// Mitsubishi GX Works2 project: Trim_Press 20-08-2023_fr   PLC: Q03UDV

PROGRAM MAIN
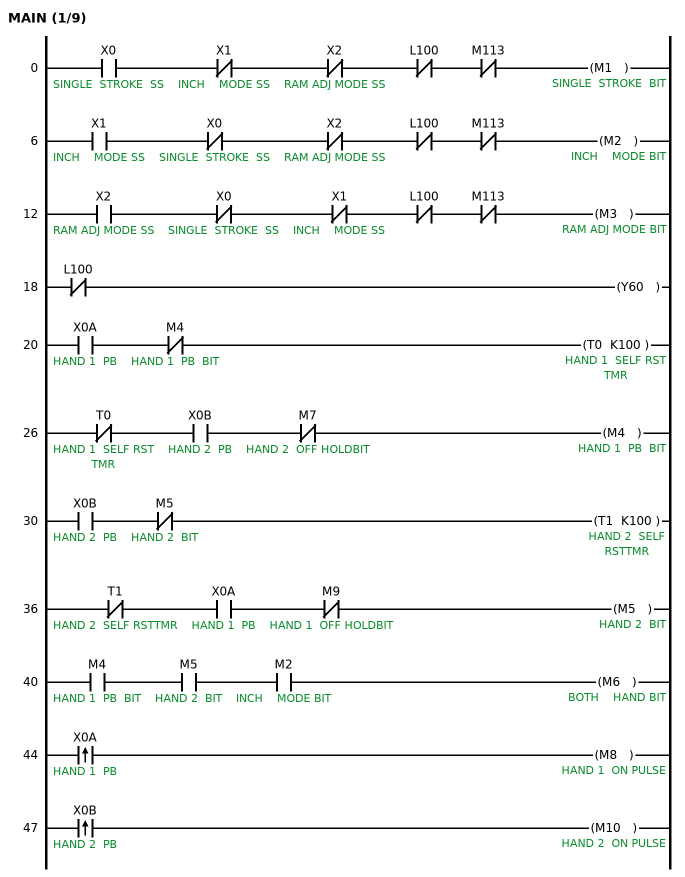
0     LD      X0  ; SINGLE  STROKE  SS
      ANI     X1  ; INCH    MODE SS
      ANI     X2  ; RAM ADJ MODE SS
      ANI     L100
      ANI     M113
      OUT     M1  ; SINGLE  STROKE  BIT
6     LD      X1  ; INCH    MODE SS
      ANI     X0  ; SINGLE  STROKE  SS
      ANI     X2  ; RAM ADJ MODE SS
      ANI     L100
      ANI     M113
      OUT     M2  ; INCH    MODE BIT
12    LD      X2  ; RAM ADJ MODE SS
      ANI     X0  ; SINGLE  STROKE  SS
      ANI     X1  ; INCH    MODE SS
      ANI     L100
      ANI     M113
      OUT     M3  ; RAM ADJ MODE BIT
18    LDI     L100
      OUT     Y60
20    LD      X0A  ; HAND 1  PB
      ANI     M4  ; HAND 1  PB  BIT
      OUT     T0 K100  ; HAND 1  SELF RST TMR
26    LDI     T0  ; HAND 1  SELF RST TMR
      AND     X0B  ; HAND 2  PB
      ANI     M7  ; HAND 2  OFF HOLDBIT
      OUT     M4  ; HAND 1  PB  BIT
30    LD      X0B  ; HAND 2  PB
      ANI     M5  ; HAND 2  BIT
      OUT     T1 K100  ; HAND 2  SELF RSTTMR
36    LDI     T1  ; HAND 2  SELF RSTTMR
      AND     X0A  ; HAND 1  PB
      ANI     M9  ; HAND 1  OFF HOLDBIT
      OUT     M5  ; HAND 2  BIT
40    LD      M4  ; HAND 1  PB  BIT
      AND     M5  ; HAND 2  BIT
      AND     M2  ; INCH    MODE BIT
      OUT     M6  ; BOTH    HAND BIT
44    LDP     X0A  ; HAND 1  PB
      OUT     M8  ; HAND 1  ON PULSE
47    LDP     X0B  ; HAND 2  PB
      OUT     M10  ; HAND 2  ON PULSE
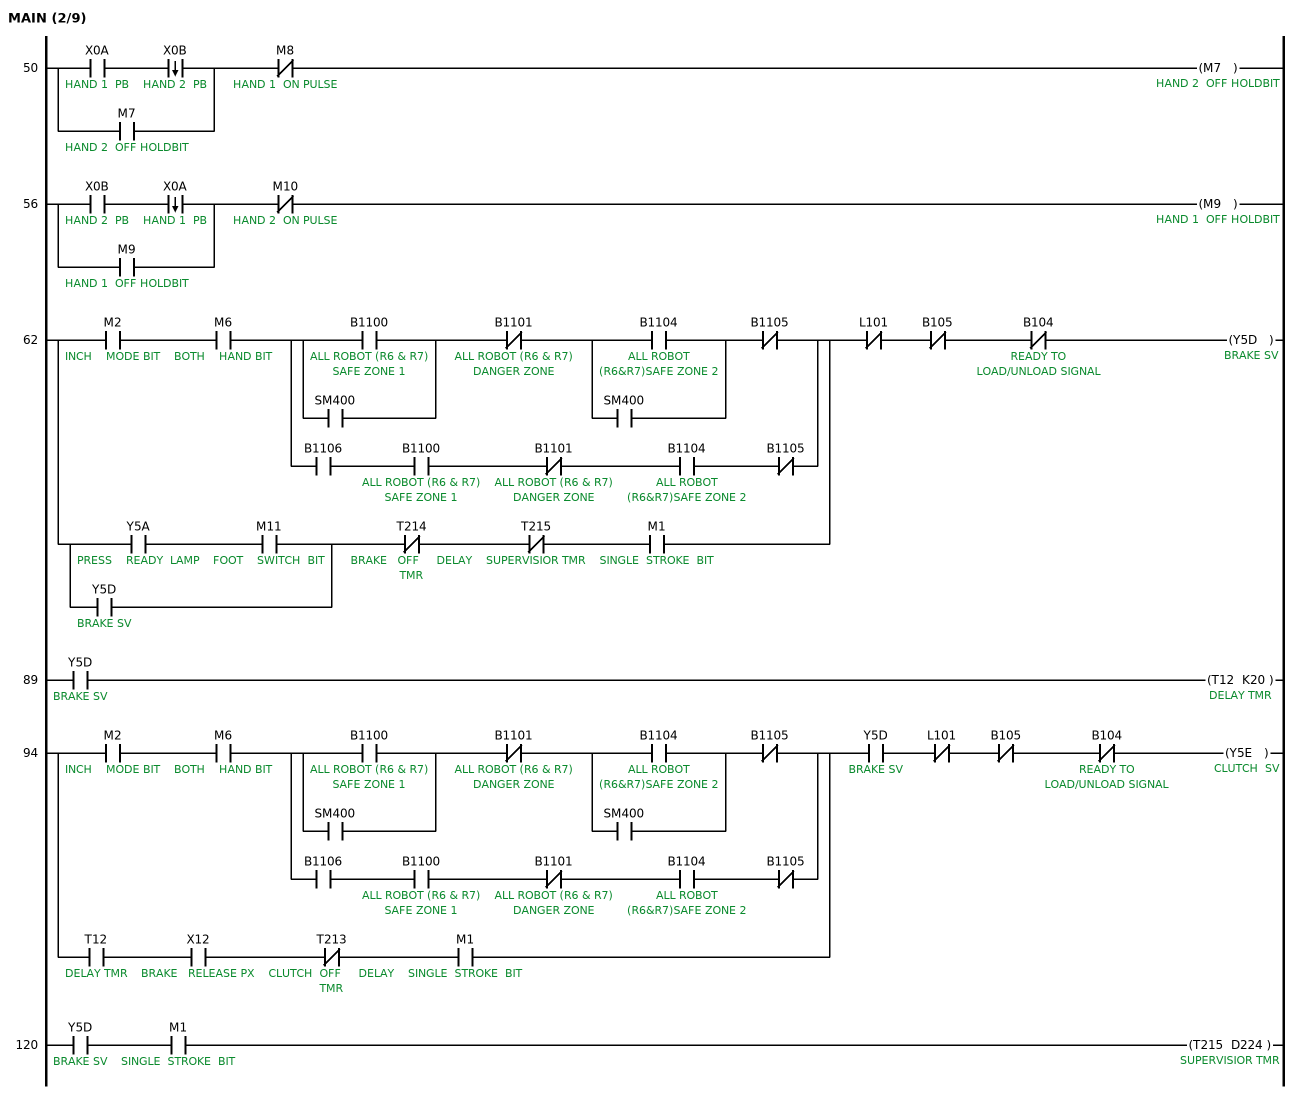
50    LD      X0A  ; HAND 1  PB
      ANDF    X0B  ; HAND 2  PB
      OR      M7  ; HAND 2  OFF HOLDBIT
      ANI     M8  ; HAND 1  ON PULSE
      OUT     M7  ; HAND 2  OFF HOLDBIT
56    LD      X0B  ; HAND 2  PB
      ANDF    X0A  ; HAND 1  PB
      OR      M9  ; HAND 1  OFF HOLDBIT
      ANI     M10  ; HAND 2  ON PULSE
      OUT     M9  ; HAND 1  OFF HOLDBIT
62    LD      M2  ; INCH    MODE BIT
      AND     M6  ; BOTH    HAND BIT
      LD      B1100  ; ALL ROBOT (R6 & R7) SAFE ZONE 1
      OR      SM400
      ANI     B1101  ; ALL ROBOT (R6 & R7) DANGER ZONE
      LD      B1104  ; ALL ROBOT (R6&R7)SAFE ZONE 2
      OR      SM400
      ANB
      ANI     B1105
      LD      B1106
      AND     B1100  ; ALL ROBOT (R6 & R7) SAFE ZONE 1
      ANI     B1101  ; ALL ROBOT (R6 & R7) DANGER ZONE
      AND     B1104  ; ALL ROBOT (R6&R7)SAFE ZONE 2
      ANI     B1105
      ORB
      ANB
      LD      Y5A  ; PRESS    READY  LAMP
      AND     M11  ; FOOT    SWITCH  BIT
      OR      Y5D  ; BRAKE SV
      ANI     T214  ; BRAKE   OFF     DELAY   TMR
      ANI     T215  ; SUPERVISIOR TMR
      AND     M1  ; SINGLE  STROKE  BIT
      ORB
      ANI     L101
      ANI     B105
      ANI     B104  ; READY TO LOAD/UNLOAD SIGNAL
      OUT     Y5D  ; BRAKE SV
89    LD      Y5D  ; BRAKE SV
      OUT     T12 K20  ; DELAY TMR
94    LD      M2  ; INCH    MODE BIT
      AND     M6  ; BOTH    HAND BIT
      LD      B1100  ; ALL ROBOT (R6 & R7) SAFE ZONE 1
      OR      SM400
      ANI     B1101  ; ALL ROBOT (R6 & R7) DANGER ZONE
      LD      B1104  ; ALL ROBOT (R6&R7)SAFE ZONE 2
      OR      SM400
      ANB
      ANI     B1105
      LD      B1106
      AND     B1100  ; ALL ROBOT (R6 & R7) SAFE ZONE 1
      ANI     B1101  ; ALL ROBOT (R6 & R7) DANGER ZONE
      AND     B1104  ; ALL ROBOT (R6&R7)SAFE ZONE 2
      ANI     B1105
      ORB
      ANB
      LD      T12  ; DELAY TMR
      AND     X12  ; BRAKE   RELEASE PX
      ANI     T213  ; CLUTCH  OFF     DELAY   TMR
      AND     M1  ; SINGLE  STROKE  BIT
      ORB
      AND     Y5D  ; BRAKE SV
      ANI     L101
      ANI     B105
      ANI     B104  ; READY TO LOAD/UNLOAD SIGNAL
      OUT     Y5E  ; CLUTCH  SV
120   LD      Y5D  ; BRAKE SV
      AND     M1  ; SINGLE  STROKE  BIT
      OUT     T215 D224  ; SUPERVISIOR TMR
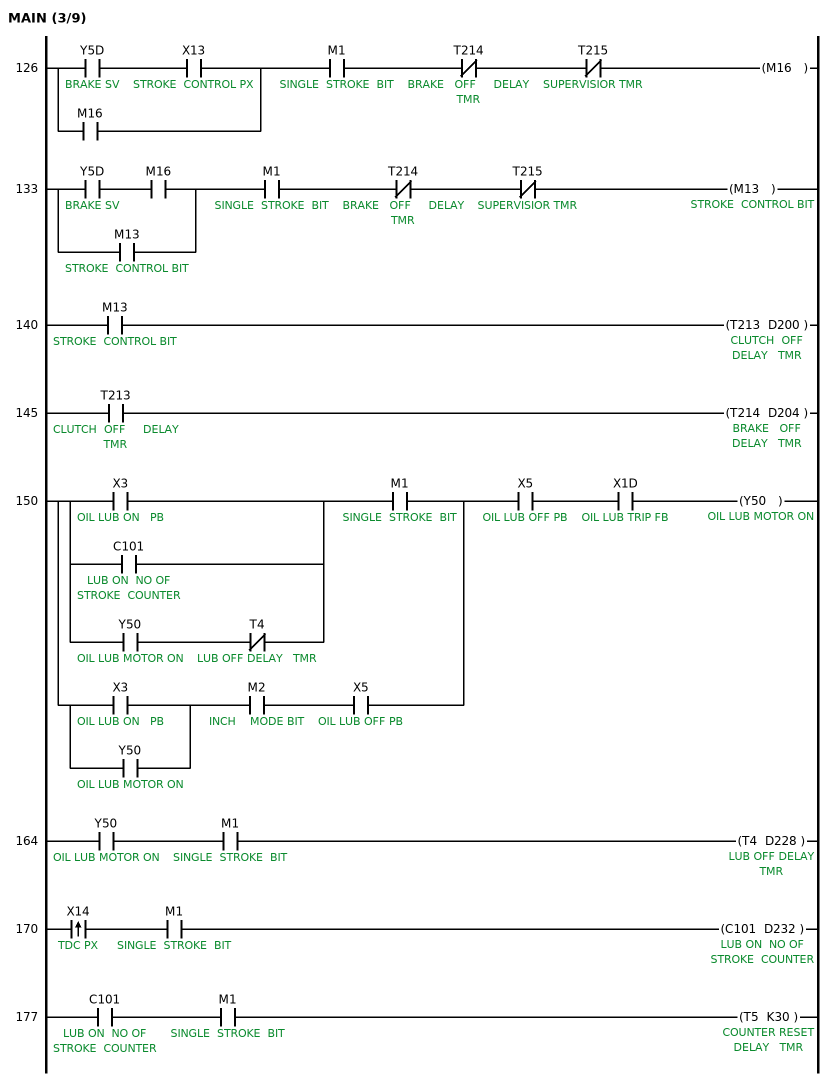
126   LD      Y5D  ; BRAKE SV
      AND     X13  ; STROKE  CONTROL PX
      OR      M16
      AND     M1  ; SINGLE  STROKE  BIT
      ANI     T214  ; BRAKE   OFF     DELAY   TMR
      ANI     T215  ; SUPERVISIOR TMR
      OUT     M16
133   LD      Y5D  ; BRAKE SV
      AND     M16
      OR      M13  ; STROKE  CONTROL BIT
      AND     M1  ; SINGLE  STROKE  BIT
      ANI     T214  ; BRAKE   OFF     DELAY   TMR
      ANI     T215  ; SUPERVISIOR TMR
      OUT     M13  ; STROKE  CONTROL BIT
140   LD      M13  ; STROKE  CONTROL BIT
      OUT     T213 D200  ; CLUTCH  OFF     DELAY   TMR
145   LD      T213  ; CLUTCH  OFF     DELAY   TMR
      OUT     T214 D204  ; BRAKE   OFF     DELAY   TMR
150   LD      X3  ; OIL LUB ON   PB
      OR      C101  ; LUB ON  NO OF   STROKE  COUNTER
      LD      Y50  ; OIL LUB MOTOR ON
      ANI     T4  ; LUB OFF DELAY   TMR
      ORB
      AND     M1  ; SINGLE  STROKE  BIT
      LD      X3  ; OIL LUB ON   PB
      OR      Y50  ; OIL LUB MOTOR ON
      AND     M2  ; INCH    MODE BIT
      AND     X5  ; OIL LUB OFF PB
      ORB
      AND     X5  ; OIL LUB OFF PB
      AND     X1D  ; OIL LUB TRIP FB
      OUT     Y50  ; OIL LUB MOTOR ON
164   LD      Y50  ; OIL LUB MOTOR ON
      AND     M1  ; SINGLE  STROKE  BIT
      OUT     T4 D228  ; LUB OFF DELAY   TMR
170   LDP     X14  ; TDC PX
      AND     M1  ; SINGLE  STROKE  BIT
      OUT     C101 D232  ; LUB ON  NO OF   STROKE  COUNTER
177   LD      C101  ; LUB ON  NO OF   STROKE  COUNTER
      AND     M1  ; SINGLE  STROKE  BIT
      OUT     T5 K30  ; COUNTER RESET   DELAY   TMR
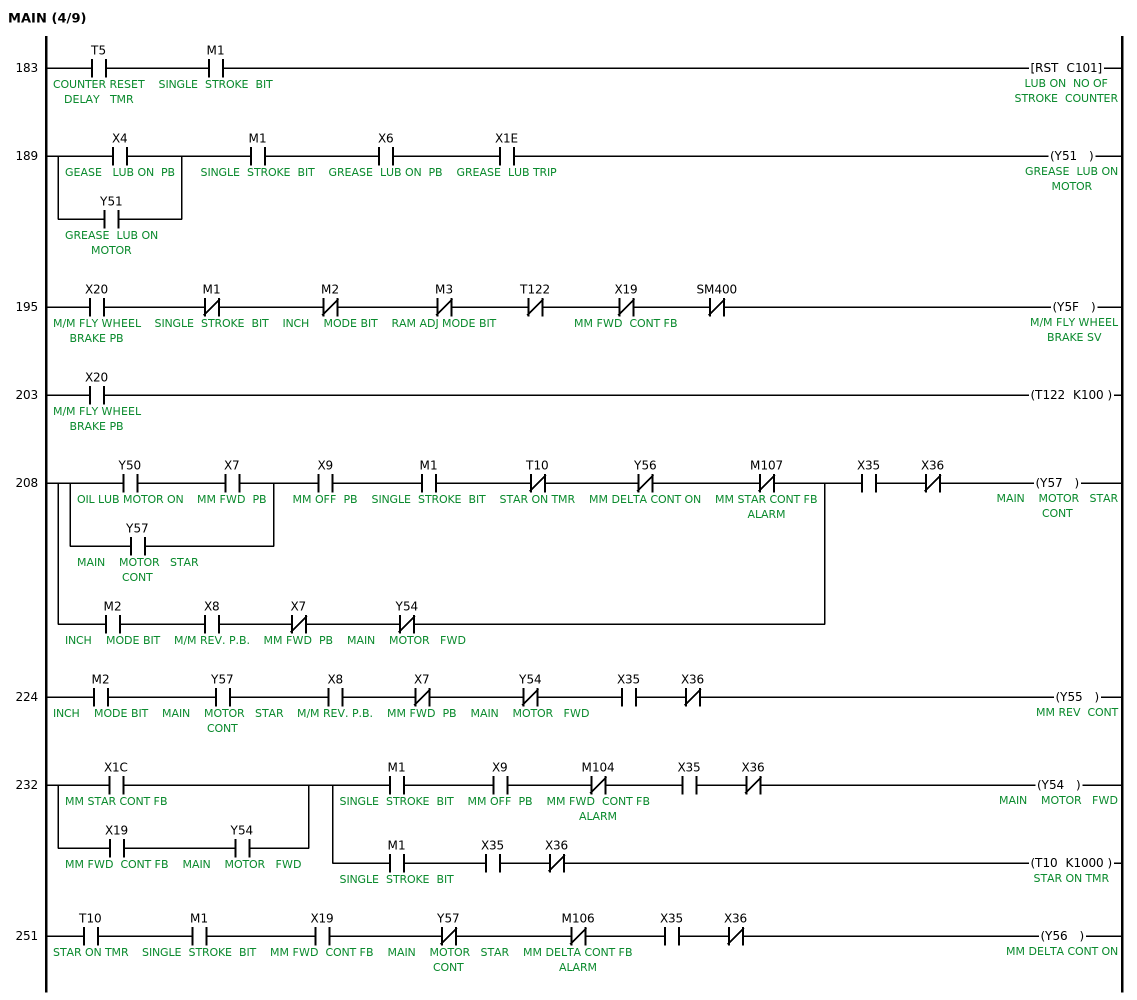
183   LD      T5  ; COUNTER RESET   DELAY   TMR
      AND     M1  ; SINGLE  STROKE  BIT
      RST     C101  ; LUB ON  NO OF   STROKE  COUNTER
189   LD      X4  ; GEASE   LUB ON  PB
      OR      Y51  ; GREASE  LUB ON   MOTOR
      AND     M1  ; SINGLE  STROKE  BIT
      AND     X6  ; GREASE  LUB ON  PB
      AND     X1E  ; GREASE  LUB TRIP
      OUT     Y51  ; GREASE  LUB ON   MOTOR
195   LD      X20  ; M/M FLY WHEEL   BRAKE PB
      ANI     M1  ; SINGLE  STROKE  BIT
      ANI     M2  ; INCH    MODE BIT
      ANI     M3  ; RAM ADJ MODE BIT
      ANI     T122
      ANI     X19  ; MM FWD  CONT FB
      ANI     SM400
      OUT     Y5F  ; M/M FLY WHEEL   BRAKE SV
203   LD      X20  ; M/M FLY WHEEL   BRAKE PB
      OUT     T122 K100
208   LD      Y50  ; OIL LUB MOTOR ON
      AND     X7  ; MM FWD  PB
      OR      Y57  ; MAIN    MOTOR   STAR    CONT
      AND     X9  ; MM OFF  PB
      AND     M1  ; SINGLE  STROKE  BIT
      ANI     T10  ; STAR ON TMR
      ANI     Y56  ; MM DELTA CONT ON
      ANI     M107  ; MM STAR CONT FB ALARM
      LD      M2  ; INCH    MODE BIT
      AND     X8  ; M/M REV. P.B.
      ANI     X7  ; MM FWD  PB
      ANI     Y54  ; MAIN    MOTOR   FWD
      ORB
      AND     X35
      ANI     X36
      OUT     Y57  ; MAIN    MOTOR   STAR    CONT
224   LD      M2  ; INCH    MODE BIT
      AND     Y57  ; MAIN    MOTOR   STAR    CONT
      AND     X8  ; M/M REV. P.B.
      ANI     X7  ; MM FWD  PB
      ANI     Y54  ; MAIN    MOTOR   FWD
      AND     X35
      ANI     X36
      OUT     Y55  ; MM REV  CONT
232   LD      X1C  ; MM STAR CONT FB
      LD      X19  ; MM FWD  CONT FB
      AND     Y54  ; MAIN    MOTOR   FWD
      ORB
      MPS
      AND     M1  ; SINGLE  STROKE  BIT
      AND     X9  ; MM OFF  PB
      ANI     M104  ; MM FWD  CONT FB  ALARM
      AND     X35
      ANI     X36
      OUT     Y54  ; MAIN    MOTOR   FWD
      MPP
      AND     M1  ; SINGLE  STROKE  BIT
      AND     X35
      ANI     X36
      OUT     T10 K1000  ; STAR ON TMR
251   LD      T10  ; STAR ON TMR
      AND     M1  ; SINGLE  STROKE  BIT
      AND     X19  ; MM FWD  CONT FB
      ANI     Y57  ; MAIN    MOTOR   STAR    CONT
      ANI     M106  ; MM DELTA CONT FB ALARM
      AND     X35
      ANI     X36
      OUT     Y56  ; MM DELTA CONT ON
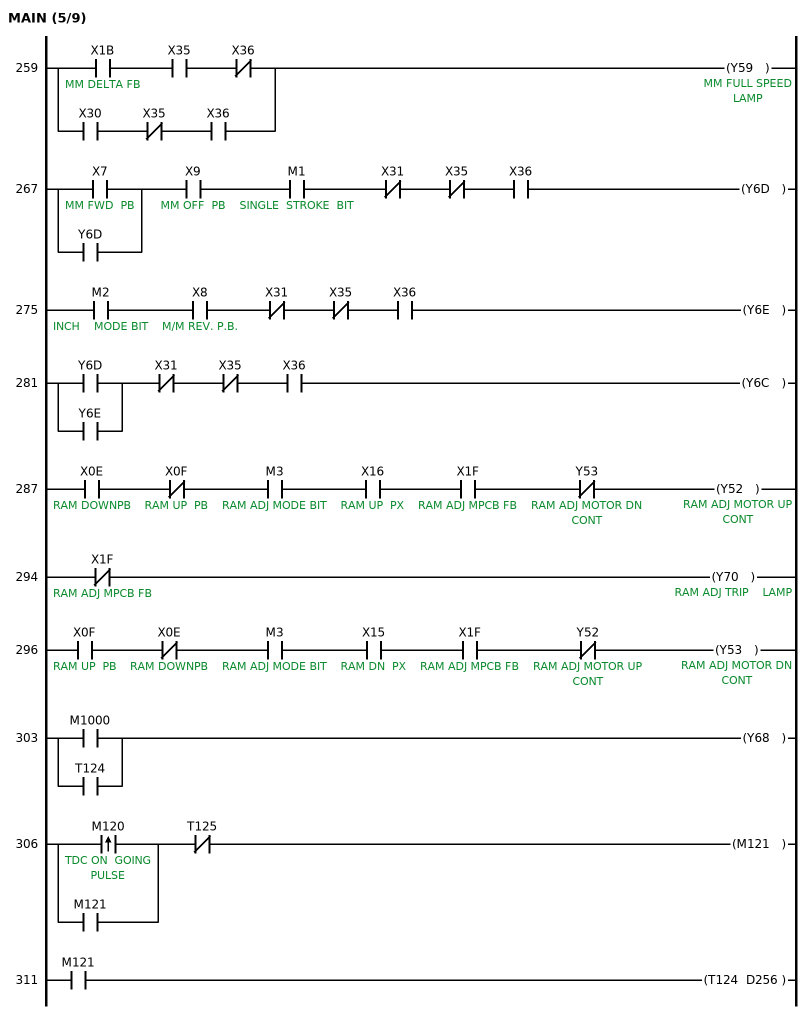
259   LD      X1B  ; MM DELTA FB
      AND     X35
      ANI     X36
      LD      X30
      ANI     X35
      AND     X36
      ORB
      OUT     Y59  ; MM FULL SPEED   LAMP
267   LD      X7  ; MM FWD  PB
      OR      Y6D
      AND     X9  ; MM OFF  PB
      AND     M1  ; SINGLE  STROKE  BIT
      ANI     X31
      ANI     X35
      AND     X36
      OUT     Y6D
275   LD      M2  ; INCH    MODE BIT
      AND     X8  ; M/M REV. P.B.
      ANI     X31
      ANI     X35
      AND     X36
      OUT     Y6E
281   LD      Y6D
      OR      Y6E
      ANI     X31
      ANI     X35
      AND     X36
      OUT     Y6C
287   LD      X0E  ; RAM DOWNPB
      ANI     X0F  ; RAM UP  PB
      AND     M3  ; RAM ADJ MODE BIT
      AND     X16  ; RAM UP  PX
      AND     X1F  ; RAM ADJ MPCB FB
      ANI     Y53  ; RAM ADJ MOTOR DN CONT
      OUT     Y52  ; RAM ADJ MOTOR UP CONT
294   LDI     X1F  ; RAM ADJ MPCB FB
      OUT     Y70  ; RAM ADJ TRIP    LAMP
296   LD      X0F  ; RAM UP  PB
      ANI     X0E  ; RAM DOWNPB
      AND     M3  ; RAM ADJ MODE BIT
      AND     X15  ; RAM DN  PX
      AND     X1F  ; RAM ADJ MPCB FB
      ANI     Y52  ; RAM ADJ MOTOR UP CONT
      OUT     Y53  ; RAM ADJ MOTOR DN CONT
303   LD      M1000
      OR      T124
      OUT     Y68
306   LDP     M120  ; TDC ON  GOING   PULSE
      OR      M121
      ANI     T125
      OUT     M121
311   LD      M121
      OUT     T124 D256
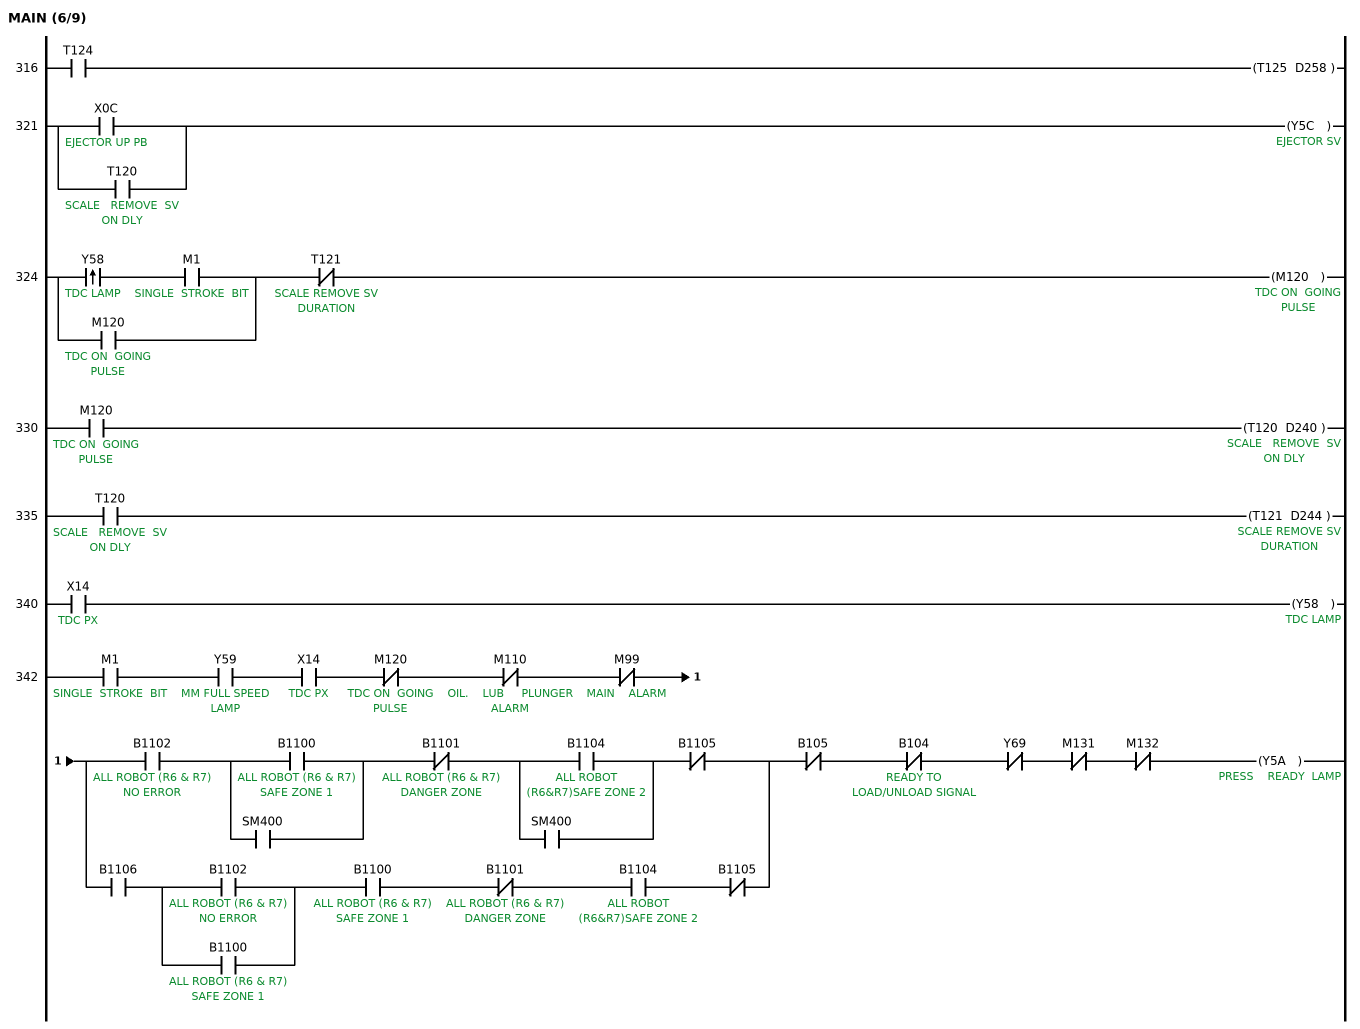
316   LD      T124
      OUT     T125 D258
321   LD      X0C  ; EJECTOR UP PB
      OR      T120  ; SCALE   REMOVE  SV   ON DLY
      OUT     Y5C  ; EJECTOR SV
324   LDP     Y58  ; TDC LAMP
      AND     M1  ; SINGLE  STROKE  BIT
      OR      M120  ; TDC ON  GOING   PULSE
      ANI     T121  ; SCALE REMOVE SV DURATION
      OUT     M120  ; TDC ON  GOING   PULSE
330   LD      M120  ; TDC ON  GOING   PULSE
      OUT     T120 D240  ; SCALE   REMOVE  SV   ON DLY
335   LD      T120  ; SCALE   REMOVE  SV   ON DLY
      OUT     T121 D244  ; SCALE REMOVE SV DURATION
340   LD      X14  ; TDC PX
      OUT     Y58  ; TDC LAMP
342   LD      M1  ; SINGLE  STROKE  BIT
      AND     Y59  ; MM FULL SPEED   LAMP
      AND     X14  ; TDC PX
      ANI     M120  ; TDC ON  GOING   PULSE
      ANI     M110  ; OIL.    LUB     PLUNGER ALARM
      ANI     M99  ; MAIN    ALARM
      LD      B1102  ; ALL ROBOT (R6 & R7) NO ERROR
      LD      B1100  ; ALL ROBOT (R6 & R7) SAFE ZONE 1
      OR      SM400
      ANB
      ANI     B1101  ; ALL ROBOT (R6 & R7) DANGER ZONE
      LD      B1104  ; ALL ROBOT (R6&R7)SAFE ZONE 2
      OR      SM400
      ANB
      ANI     B1105
      LD      B1106
      LD      B1102  ; ALL ROBOT (R6 & R7) NO ERROR
      OR      B1100  ; ALL ROBOT (R6 & R7) SAFE ZONE 1
      ANB
      AND     B1100  ; ALL ROBOT (R6 & R7) SAFE ZONE 1
      ANI     B1101  ; ALL ROBOT (R6 & R7) DANGER ZONE
      AND     B1104  ; ALL ROBOT (R6&R7)SAFE ZONE 2
      ANI     B1105
      ORB
      ANB
      ANI     B105
      ANI     B104  ; READY TO LOAD/UNLOAD SIGNAL
      ANI     Y69
      ANI     M131
      ANI     M132
      OUT     Y5A  ; PRESS    READY  LAMP
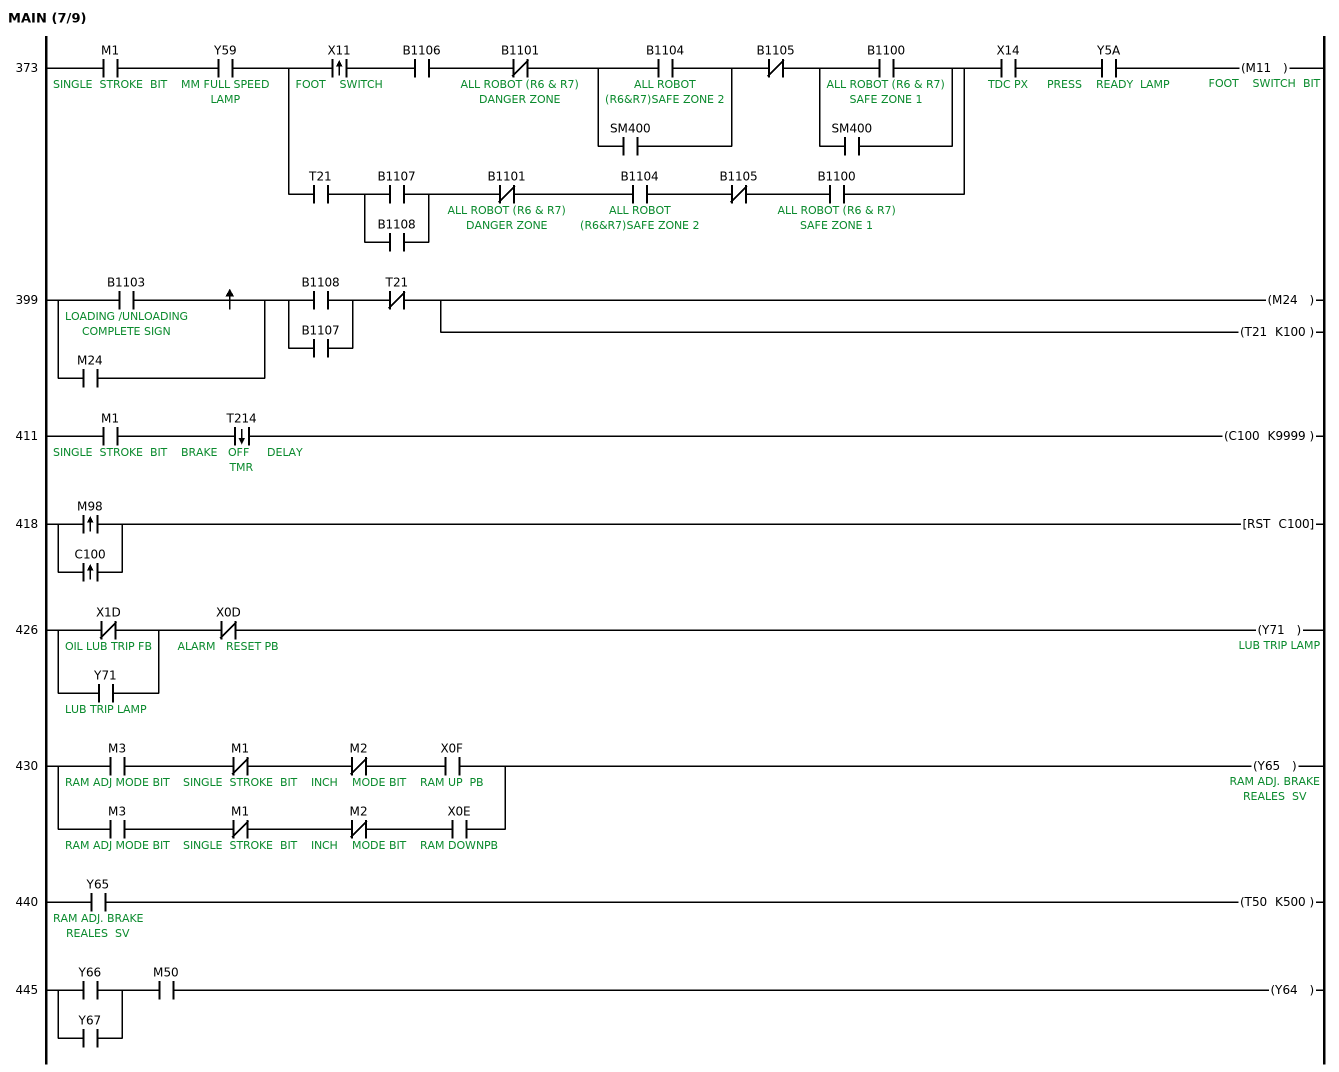
373   LD      M1  ; SINGLE  STROKE  BIT
      AND     Y59  ; MM FULL SPEED   LAMP
      LDP     X11  ; FOOT    SWITCH
      AND     B1106
      ANI     B1101  ; ALL ROBOT (R6 & R7) DANGER ZONE
      LD      B1104  ; ALL ROBOT (R6&R7)SAFE ZONE 2
      OR      SM400
      ANB
      ANI     B1105
      LD      B1100  ; ALL ROBOT (R6 & R7) SAFE ZONE 1
      OR      SM400
      ANB
      LD      T21
      LD      B1107
      OR      B1108
      ANB
      ANI     B1101  ; ALL ROBOT (R6 & R7) DANGER ZONE
      AND     B1104  ; ALL ROBOT (R6&R7)SAFE ZONE 2
      ANI     B1105
      AND     B1100  ; ALL ROBOT (R6 & R7) SAFE ZONE 1
      ORB
      ANB
      AND     X14  ; TDC PX
      AND     Y5A  ; PRESS    READY  LAMP
      OUT     M11  ; FOOT    SWITCH  BIT
399   LD      B1103  ; LOADING /UNLOADING COMPLETE SIGN
      MEP
      OR      M24
      LD      B1108
      OR      B1107
      ANB
      ANI     T21
      OUT     M24
      OUT     T21 K100
411   LD      M1  ; SINGLE  STROKE  BIT
      ANDF    T214  ; BRAKE   OFF     DELAY   TMR
      OUT     C100 K9999
418   LDP     M98
      ORP     C100
      RST     C100
426   LDI     X1D  ; OIL LUB TRIP FB
      OR      Y71  ; LUB TRIP LAMP
      ANI     X0D  ; ALARM   RESET PB
      OUT     Y71  ; LUB TRIP LAMP
430   LD      M3  ; RAM ADJ MODE BIT
      ANI     M1  ; SINGLE  STROKE  BIT
      ANI     M2  ; INCH    MODE BIT
      AND     X0F  ; RAM UP  PB
      LD      M3  ; RAM ADJ MODE BIT
      ANI     M1  ; SINGLE  STROKE  BIT
      ANI     M2  ; INCH    MODE BIT
      AND     X0E  ; RAM DOWNPB
      ORB
      OUT     Y65  ; RAM ADJ. BRAKE  REALES  SV
440   LD      Y65  ; RAM ADJ. BRAKE  REALES  SV
      OUT     T50 K500
445   LD      Y66
      OR      Y67
      AND     M50
      OUT     Y64
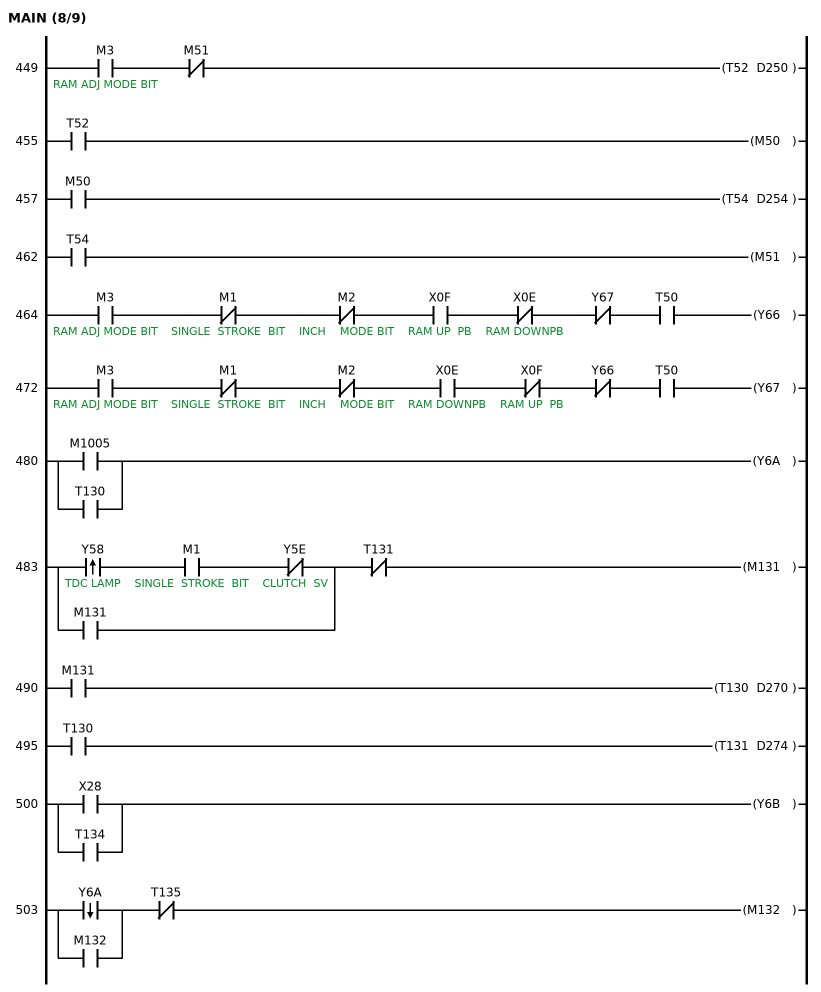
449   LD      M3  ; RAM ADJ MODE BIT
      ANI     M51
      OUT     T52 D250
455   LD      T52
      OUT     M50
457   LD      M50
      OUT     T54 D254
462   LD      T54
      OUT     M51
464   LD      M3  ; RAM ADJ MODE BIT
      ANI     M1  ; SINGLE  STROKE  BIT
      ANI     M2  ; INCH    MODE BIT
      AND     X0F  ; RAM UP  PB
      ANI     X0E  ; RAM DOWNPB
      ANI     Y67
      AND     T50
      OUT     Y66
472   LD      M3  ; RAM ADJ MODE BIT
      ANI     M1  ; SINGLE  STROKE  BIT
      ANI     M2  ; INCH    MODE BIT
      AND     X0E  ; RAM DOWNPB
      ANI     X0F  ; RAM UP  PB
      ANI     Y66
      AND     T50
      OUT     Y67
480   LD      M1005
      OR      T130
      OUT     Y6A
483   LDP     Y58  ; TDC LAMP
      AND     M1  ; SINGLE  STROKE  BIT
      ANI     Y5E  ; CLUTCH  SV
      OR      M131
      ANI     T131
      OUT     M131
490   LD      M131
      OUT     T130 D270
495   LD      T130
      OUT     T131 D274
500   LD      X28
      OR      T134
      OUT     Y6B
503   LDF     Y6A
      OR      M132
      ANI     T135
      OUT     M132
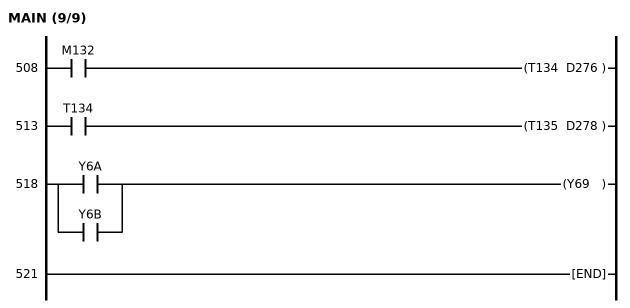
508   LD      M132
      OUT     T134 D276
513   LD      T134
      OUT     T135 D278
518   LD      Y6A
      OR      Y6B
      OUT     Y69
521   END
END_PROGRAM

PROGRAM MAIN01
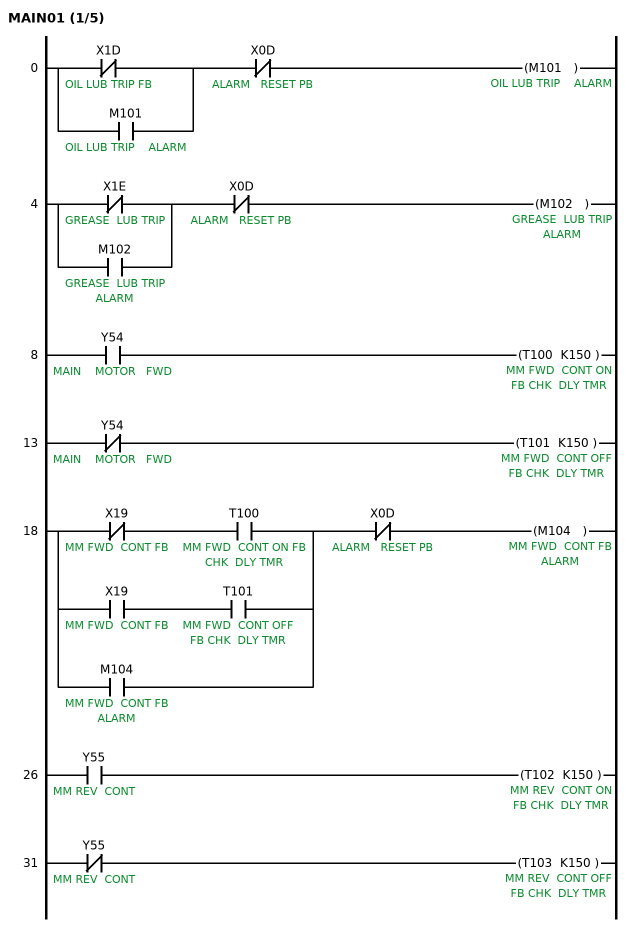
0     LDI     X1D  ; OIL LUB TRIP FB
      OR      M101  ; OIL LUB TRIP    ALARM
      ANI     X0D  ; ALARM   RESET PB
      OUT     M101  ; OIL LUB TRIP    ALARM
4     LDI     X1E  ; GREASE  LUB TRIP
      OR      M102  ; GREASE  LUB TRIP  ALARM
      ANI     X0D  ; ALARM   RESET PB
      OUT     M102  ; GREASE  LUB TRIP  ALARM
8     LD      Y54  ; MAIN    MOTOR   FWD
      OUT     T100 K150  ; MM FWD  CONT ON FB CHK  DLY TMR
13    LDI     Y54  ; MAIN    MOTOR   FWD
      OUT     T101 K150  ; MM FWD  CONT OFF FB CHK  DLY TMR
18    LDI     X19  ; MM FWD  CONT FB
      AND     T100  ; MM FWD  CONT ON FB CHK  DLY TMR
      LD      X19  ; MM FWD  CONT FB
      AND     T101  ; MM FWD  CONT OFF FB CHK  DLY TMR
      ORB
      OR      M104  ; MM FWD  CONT FB  ALARM
      ANI     X0D  ; ALARM   RESET PB
      OUT     M104  ; MM FWD  CONT FB  ALARM
26    LD      Y55  ; MM REV  CONT
      OUT     T102 K150  ; MM REV  CONT ON FB CHK  DLY TMR
31    LDI     Y55  ; MM REV  CONT
      OUT     T103 K150  ; MM REV  CONT OFF FB CHK  DLY TMR
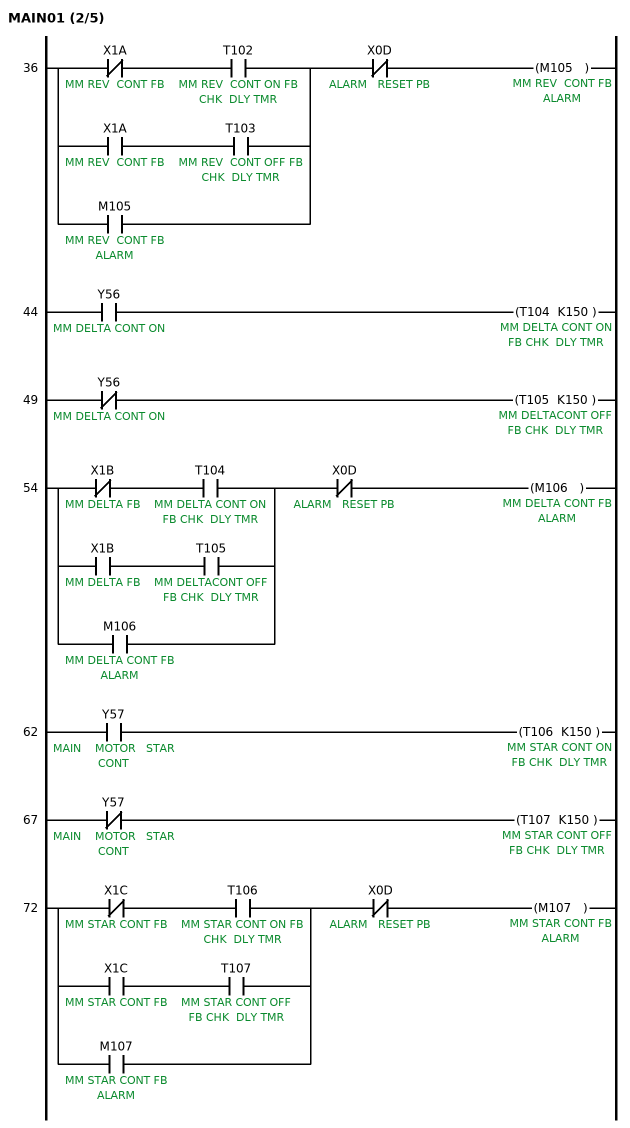
36    LDI     X1A  ; MM REV  CONT FB
      AND     T102  ; MM REV  CONT ON FB CHK  DLY TMR
      LD      X1A  ; MM REV  CONT FB
      AND     T103  ; MM REV  CONT OFF FB CHK  DLY TMR
      ORB
      OR      M105  ; MM REV  CONT FB ALARM
      ANI     X0D  ; ALARM   RESET PB
      OUT     M105  ; MM REV  CONT FB ALARM
44    LD      Y56  ; MM DELTA CONT ON
      OUT     T104 K150  ; MM DELTA CONT ON FB CHK  DLY TMR
49    LDI     Y56  ; MM DELTA CONT ON
      OUT     T105 K150  ; MM DELTACONT OFF FB CHK  DLY TMR
54    LDI     X1B  ; MM DELTA FB
      AND     T104  ; MM DELTA CONT ON FB CHK  DLY TMR
      LD      X1B  ; MM DELTA FB
      AND     T105  ; MM DELTACONT OFF FB CHK  DLY TMR
      ORB
      OR      M106  ; MM DELTA CONT FB ALARM
      ANI     X0D  ; ALARM   RESET PB
      OUT     M106  ; MM DELTA CONT FB ALARM
62    LD      Y57  ; MAIN    MOTOR   STAR    CONT
      OUT     T106 K150  ; MM STAR CONT ON FB CHK  DLY TMR
67    LDI     Y57  ; MAIN    MOTOR   STAR    CONT
      OUT     T107 K150  ; MM STAR CONT OFF FB CHK  DLY TMR
72    LDI     X1C  ; MM STAR CONT FB
      AND     T106  ; MM STAR CONT ON FB CHK  DLY TMR
      LD      X1C  ; MM STAR CONT FB
      AND     T107  ; MM STAR CONT OFF FB CHK  DLY TMR
      ORB
      OR      M107  ; MM STAR CONT FB ALARM
      ANI     X0D  ; ALARM   RESET PB
      OUT     M107  ; MM STAR CONT FB ALARM
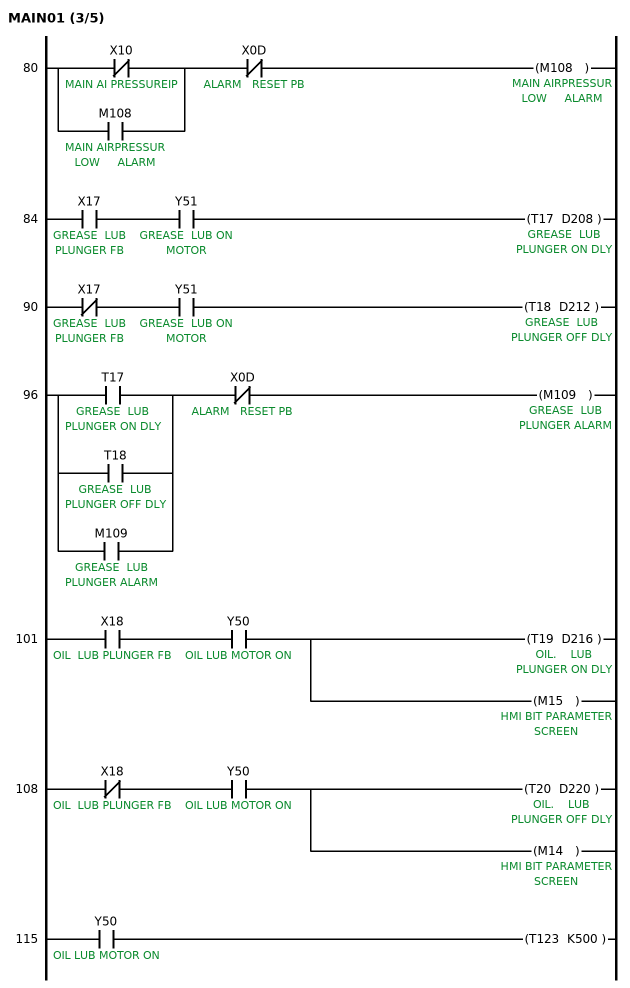
80    LDI     X10  ; MAIN AI PRESSUREIP
      OR      M108  ; MAIN AIRPRESSUR LOW     ALARM
      ANI     X0D  ; ALARM   RESET PB
      OUT     M108  ; MAIN AIRPRESSUR LOW     ALARM
84    LD      X17  ; GREASE  LUB     PLUNGER FB
      AND     Y51  ; GREASE  LUB ON   MOTOR
      OUT     T17 D208  ; GREASE  LUB     PLUNGER ON DLY
90    LDI     X17  ; GREASE  LUB     PLUNGER FB
      AND     Y51  ; GREASE  LUB ON   MOTOR
      OUT     T18 D212  ; GREASE  LUB     PLUNGER OFF DLY
96    LD      T17  ; GREASE  LUB     PLUNGER ON DLY
      OR      T18  ; GREASE  LUB     PLUNGER OFF DLY
      OR      M109  ; GREASE  LUB     PLUNGER ALARM
      ANI     X0D  ; ALARM   RESET PB
      OUT     M109  ; GREASE  LUB     PLUNGER ALARM
101   LD      X18  ; OIL  LUB PLUNGER FB
      AND     Y50  ; OIL LUB MOTOR ON
      OUT     T19 D216  ; OIL.    LUB     PLUNGER ON DLY
      OUT     M15  ; HMI BIT PARAMETER SCREEN
108   LDI     X18  ; OIL  LUB PLUNGER FB
      AND     Y50  ; OIL LUB MOTOR ON
      OUT     T20 D220  ; OIL.    LUB     PLUNGER OFF DLY
      OUT     M14  ; HMI BIT PARAMETER SCREEN
115   LD      Y50  ; OIL LUB MOTOR ON
      OUT     T123 K500
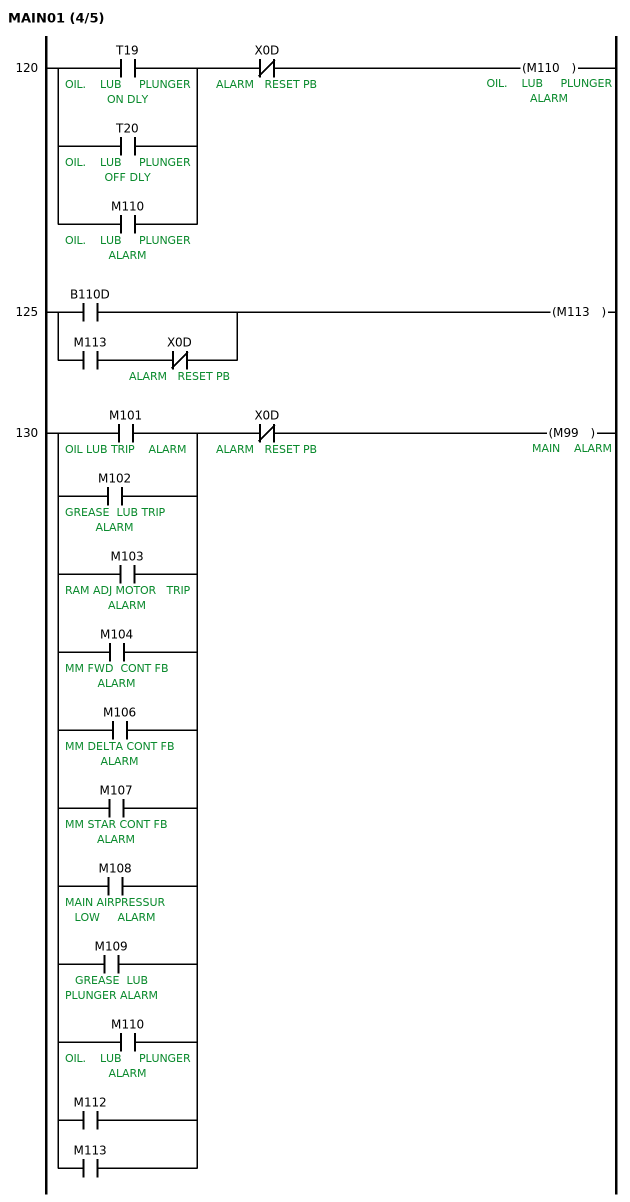
120   LD      T19  ; OIL.    LUB     PLUNGER ON DLY
      OR      T20  ; OIL.    LUB     PLUNGER OFF DLY
      OR      M110  ; OIL.    LUB     PLUNGER ALARM
      ANI     X0D  ; ALARM   RESET PB
      OUT     M110  ; OIL.    LUB     PLUNGER ALARM
125   LD      B110D
      LD      M113
      ANI     X0D  ; ALARM   RESET PB
      ORB
      OUT     M113
130   LD      M101  ; OIL LUB TRIP    ALARM
      OR      M102  ; GREASE  LUB TRIP  ALARM
      OR      M103  ; RAM ADJ MOTOR   TRIP    ALARM
      OR      M104  ; MM FWD  CONT FB  ALARM
      OR      M106  ; MM DELTA CONT FB ALARM
      OR      M107  ; MM STAR CONT FB ALARM
      OR      M108  ; MAIN AIRPRESSUR LOW     ALARM
      OR      M109  ; GREASE  LUB     PLUNGER ALARM
      OR      M110  ; OIL.    LUB     PLUNGER ALARM
      OR      M112
      OR      M113
      ANI     X0D  ; ALARM   RESET PB
      OUT     M99  ; MAIN    ALARM
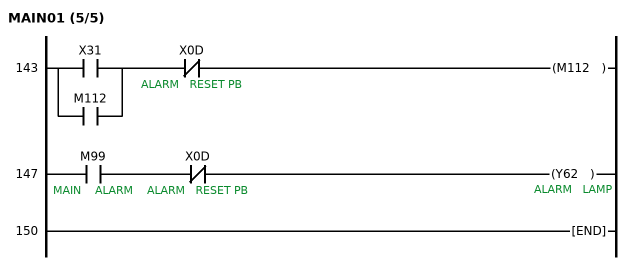
143   LD      X31
      OR      M112
      ANI     X0D  ; ALARM   RESET PB
      OUT     M112
147   LD      M99  ; MAIN    ALARM
      ANI     X0D  ; ALARM   RESET PB
      OUT     Y62  ; ALARM   LAMP
150   END
END_PROGRAM

PROGRAM R6_R7_AU
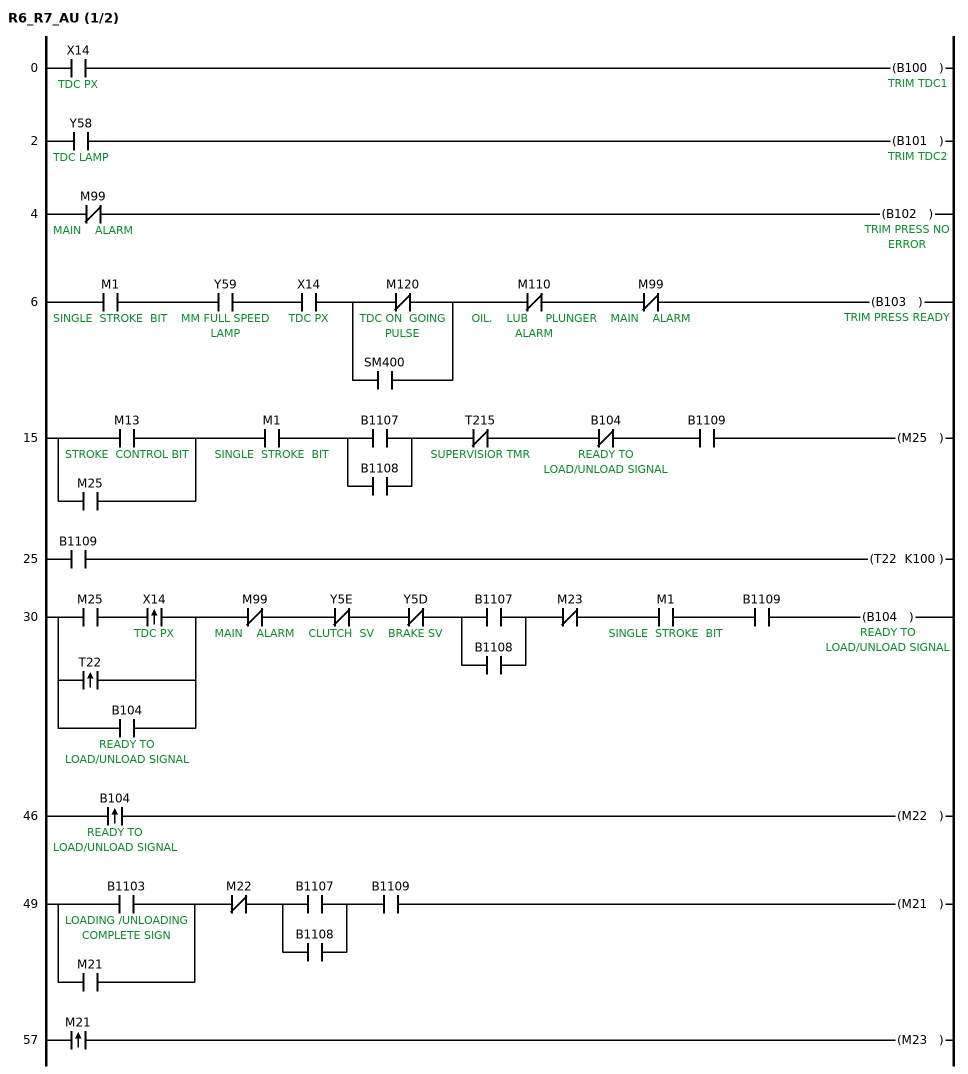
0     LD      X14  ; TDC PX
      OUT     B100  ; TRIM TDC1
2     LD      Y58  ; TDC LAMP
      OUT     B101  ; TRIM TDC2
4     LDI     M99  ; MAIN    ALARM
      OUT     B102  ; TRIM PRESS NO ERROR
6     LD      M1  ; SINGLE  STROKE  BIT
      AND     Y59  ; MM FULL SPEED   LAMP
      AND     X14  ; TDC PX
      LDI     M120  ; TDC ON  GOING   PULSE
      OR      SM400
      ANB
      ANI     M110  ; OIL.    LUB     PLUNGER ALARM
      ANI     M99  ; MAIN    ALARM
      OUT     B103  ; TRIM PRESS READY
15    LD      M13  ; STROKE  CONTROL BIT
      OR      M25
      AND     M1  ; SINGLE  STROKE  BIT
      LD      B1107
      OR      B1108
      ANB
      ANI     T215  ; SUPERVISIOR TMR
      ANI     B104  ; READY TO LOAD/UNLOAD SIGNAL
      AND     B1109
      OUT     M25
25    LD      B1109
      OUT     T22 K100
30    LD      M25
      ANDP    X14  ; TDC PX
      ORP     T22
      OR      B104  ; READY TO LOAD/UNLOAD SIGNAL
      ANI     M99  ; MAIN    ALARM
      ANI     Y5E  ; CLUTCH  SV
      ANI     Y5D  ; BRAKE SV
      LD      B1107
      OR      B1108
      ANB
      ANI     M23
      AND     M1  ; SINGLE  STROKE  BIT
      AND     B1109
      OUT     B104  ; READY TO LOAD/UNLOAD SIGNAL
46    LDP     B104  ; READY TO LOAD/UNLOAD SIGNAL
      OUT     M22
49    LD      B1103  ; LOADING /UNLOADING COMPLETE SIGN
      OR      M21
      ANI     M22
      LD      B1107
      OR      B1108
      ANB
      AND     B1109
      OUT     M21
57    LDP     M21
      OUT     M23
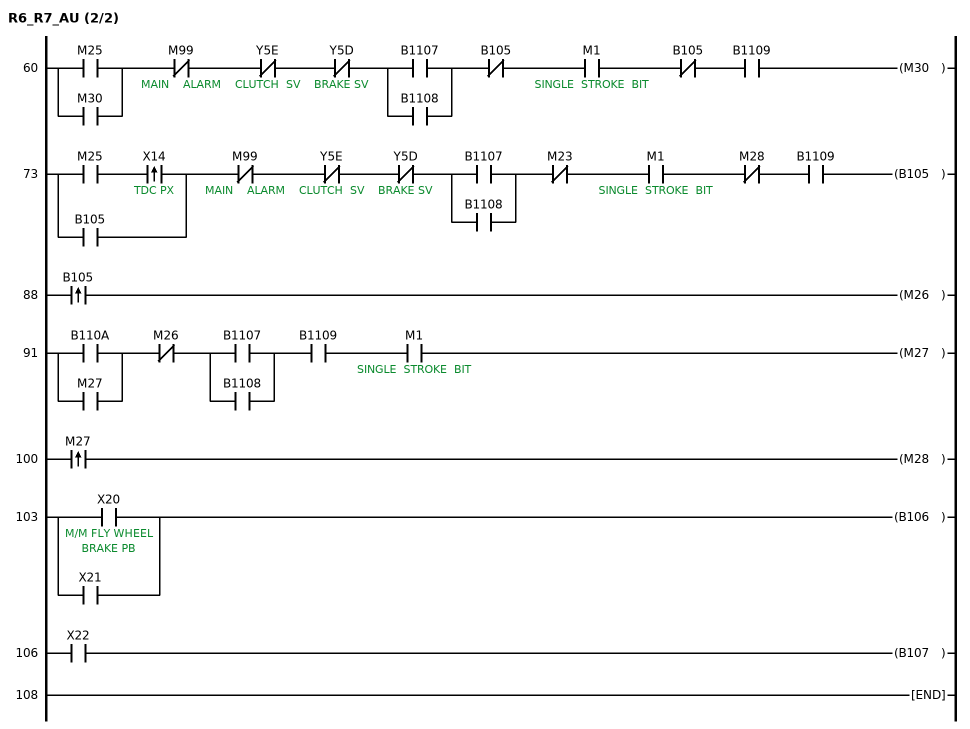
60    LD      M25
      OR      M30
      ANI     M99  ; MAIN    ALARM
      ANI     Y5E  ; CLUTCH  SV
      ANI     Y5D  ; BRAKE SV
      LD      B1107
      OR      B1108
      ANB
      ANI     B105
      AND     M1  ; SINGLE  STROKE  BIT
      ANI     B105
      AND     B1109
      OUT     M30
73    LD      M25
      ANDP    X14  ; TDC PX
      OR      B105
      ANI     M99  ; MAIN    ALARM
      ANI     Y5E  ; CLUTCH  SV
      ANI     Y5D  ; BRAKE SV
      LD      B1107
      OR      B1108
      ANB
      ANI     M23
      AND     M1  ; SINGLE  STROKE  BIT
      ANI     M28
      AND     B1109
      OUT     B105
88    LDP     B105
      OUT     M26
91    LD      B110A
      OR      M27
      ANI     M26
      LD      B1107
      OR      B1108
      ANB
      AND     B1109
      AND     M1  ; SINGLE  STROKE  BIT
      OUT     M27
100   LDP     M27
      OUT     M28
103   LD      X20  ; M/M FLY WHEEL   BRAKE PB
      OR      X21
      OUT     B106
106   LD      X22
      OUT     B107
108   END
END_PROGRAM

// device comments not shown above
M111  ; BRAKE   RELEASE PX FB   FAIL
T13  ; CLUTCH  OFF     DELAY   TMR
T14  ; BRAKE   OFF     DELAY
T15  ; SUPERVISER TMR
T108  ; BRAKE   RELEASE CHK DELAY TMR
